Fanuc KAREL source: kt00573.KL

-- PROVISIONAL review KL for V940-1; original PC SHA256 667fa695a9063174077bd8ba5a369f752a956ea19a978048fbebcc9ee81467f1
-- Incomplete behavior may be omitted. Consult companion uncertainty JSON. Do not deploy.
PROGRAM KT00573
%NOLOCKGROUP
VAR
  R1 : REAL
-- UNRESOLVED_DECL V2 type=000013
-- UNRESOLVED_DECL OUT type=000013
BEGIN
  -- V9_ZERO_TABLE_METADATA_HINT layout=0001; no indexed target words; source/name/runtime held
  -- UNRESOLVED_PC offsets 5-16; opcodes 2E,23
  -- UNRESOLVED_PC offsets 21-36; opcodes 2E,22,32,35
  -- UNRESOLVED_PC offsets 41-63; opcodes 21,49,8C,4A
  -- UNRESOLVED_PC offsets 68-72; opcodes 7F
END KT00573
